// TIA Portal V16 export
// export: Created 2023-03-29T11:03:15.4166072Z, ExportSetting WithDefaults, DisplayName Totally Integrated Automation Portal, DisplayVersion V16 Update 6, DisplayName TIA Portal Version Control Interface, DisplayVersion V16 Update 2, DisplayName TIA Portal Openness, DisplayVersion V16 Update 6, DisplayName STEP 7 Professional, DisplayVersion V16 Update 6, DisplayName STEP 7 Safety, DisplayVersion V16, DisplayName WinCC Advanced, DisplayVersion V16 Update 6
ORGANIZATION_BLOCK "Cyclic interrupt_WatchDog_comunication"   // OB32, LAD, CyclicInterrupt
TITLE = Kontrola komunikacji TCP, HMI, PLC
{ S7_Optimized_Access := 'TRUE' }
AUTHOR : rtecmer
VERSION : 0.1
// stored: AutoNumber true, IsIECCheckEnabled false, SetENOAutomatically false
   VAR_INPUT
      Initial_Call : Bool;   // Initial call of this OB
      Event_Count : Int;   // Events discarded
   END_VAR
BEGIN

REGION Network 1
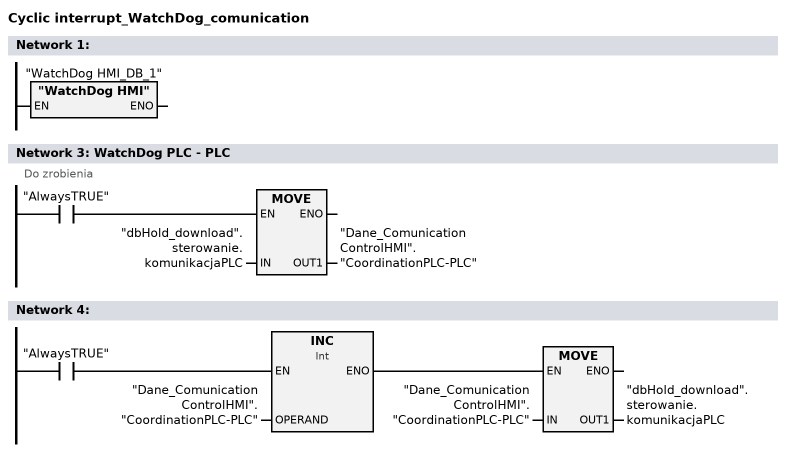
   RUNG wire#powerrail
      "WatchDog HMI_DB_1"()
   END_RUNG
   // the same network as SCL:
   "WatchDog HMI_DB_1"();   // "WatchDog HMI"
END_REGION

REGION Network 3: WatchDog PLC - PLC
   // Do zrobienia
   RUNG wire#powerrail
      Contact( "AlwaysTRUE" )
      Move(in := "dbHold_download".sterowanie.komunikacjaPLC, out1 => "Dane_ComunicationControlHMI"."CoordinationPLC-PLC")
   END_RUNG
   // the same network as SCL:
   IF "AlwaysTRUE" THEN
       "Dane_ComunicationControlHMI"."CoordinationPLC-PLC" := "dbHold_download".sterowanie.komunikacjaPLC;
   END_IF;
END_REGION

REGION Network 4
   RUNG wire#powerrail
      Contact( "AlwaysTRUE" )
      { S7_Templates := "DestType := Int" } Inc( "Dane_ComunicationControlHMI"."CoordinationPLC-PLC" )
      Move(in := "Dane_ComunicationControlHMI"."CoordinationPLC-PLC", out1 => "dbHold_download".sterowanie.komunikacjaPLC)
   END_RUNG
   // the same network as SCL:
   IF "AlwaysTRUE" THEN
       "Dane_ComunicationControlHMI"."CoordinationPLC-PLC" := "Dane_ComunicationControlHMI"."CoordinationPLC-PLC" + 1;
       "dbHold_download".sterowanie.komunikacjaPLC := "Dane_ComunicationControlHMI"."CoordinationPLC-PLC";
   END_IF;
END_REGION

REGION Network 6 (SCL): kasowanie znacznków HMI
   // znaczniki HMI do kasowania alrmów ekranów
   "dbtags_Sterowanie".HMI.resetScreen_1 := FALSE;
   "dbtags_Sterowanie".HMI.resetScreen_2 := FALSE;
   "dbtags_Sterowanie".HMI.resetScreen_3 := FALSE;
   "dbtags_Sterowanie".HMI.resetScreen_4 := FALSE;
   "dbtags_Sterowanie".HMI.resetScreen_5 := FALSE;
   "dbtags_Sterowanie".HMI.resetScreen_6 := FALSE;
   "dbtags_Sterowanie".HMI.resetScreen_7 := FALSE;
   "dbtags_Sterowanie".HMI.resetScreen_8 := FALSE;
END_REGION
END_ORGANIZATION_BLOCK
